{attribute 'GeneratedUsingTerminal: EL2212-0000-0020'}
{attribute addProperty BoxType "EL2212-0000-0020"}
{attribute addProperty Id "StatusAT %I*Status_8D3FCD237"}
{attribute addProperty CRC "1876802200"}
{attribute addProperty Size "7"}
TYPE DOX_Status_Channel_6FDDBA98 EXTENDS InputBase_8311D824 :
STRUCT
	{attribute addProperty Name "Status"}
	Status AT %I* : Status_8D3FCD23;
END_STRUCT
END_TYPE

(* stored: Version 1.2.0.0, ProductVersion 3.1.4024.9
   DUT DOX_Status_Channel_6FDDBA98: Id {7e97b68d-30ce-41ce-b540-a2d925398801} *)
